Universal Robots PolyScope program: Pick_Place_demo.urp

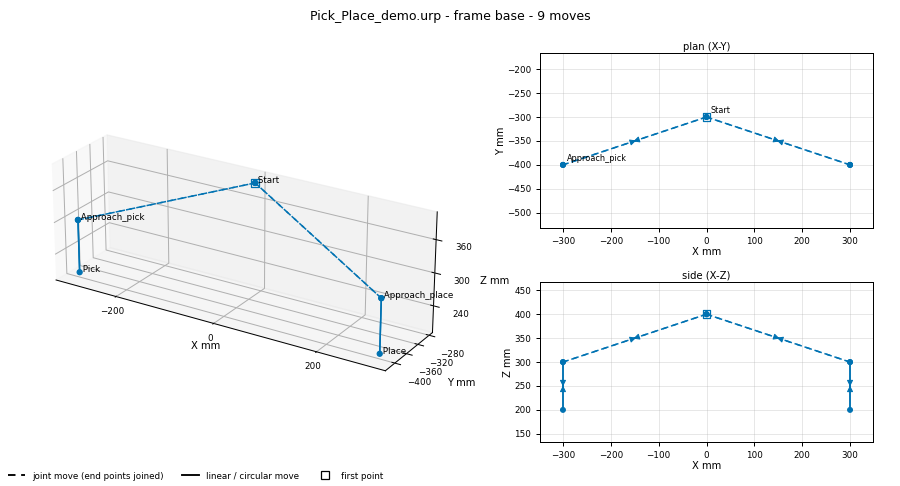
[picture p0: tool path of Pick_Place_demo.urp in frame base, 9 of 9 moves have a stored position in this frame; points joined in program order, loops and branches not executed]
Program Pick_Place_demo (installation=default directory=/programs/usbdisk createdIn=5.9.1.1031110 lastSavedIn=5.8.0.10253 robotSerialNumber=20205501179)
Calibrated DH parameters: a=[0.000177, -0.238276, -0.392216, 0.000101, -0.000031, 0]; d=[0.16274, -356.990158, 358.765662, -1.642182, 0.099681, 0.099622]; alpha=[1.570882, -0.000987, 0.009118, 1.568686, -1.570357, 0]; deltaTheta=[0, 0.976178, -0.934918, -0.041252, 0.000001, 0]
Robot Program (runOnlyOnce=false)
  MoveJ speed 60 deg/s, acceleration 80 deg/s^2 (useActiveTCP=true) feature=Base
    Waypoint Start: TCP in base x=0 y=-300 z=400 mm, rx=0 ry=3.1416 rz=0 rad; joints [-63.619, -58.456, -125.213, -86.33, 90, 26.381] deg
  Folder Pick
    MoveJ speed 60 deg/s, acceleration 80 deg/s^2 (useActiveTCP=true) feature=Base
      Waypoint Approach_pick: TCP in base x=-300 y=-400 z=300 mm, rx=0 ry=3.1416 rz=0 rad; joints [-111.408, -95.003, -113.354, -61.643, 90, -21.408] deg
    MoveL speed 250 mm/s, acceleration 1200 mm/s^2 (useActiveTCP=true) feature=Base
      Waypoint Pick: TCP in base x=-300 y=-400 z=200 mm, rx=0 ry=3.1416 rz=0 rad; joints [-111.408, -104.003, -120.574, -45.423, 90, -21.408] deg
      URCap 2FG Grip (OnRobot, OnRobot A/S) dataModel(twofg.external-grip.target-width=0.05, twofg.internal-grip.target-width=0.064, payload-weight=0.2)
      Waypoint Approach_pick: TCP in base x=-300 y=-400 z=300 mm, rx=0 ry=3.1416 rz=0 rad; joints [-111.408, -95.003, -113.354, -61.643, 90, -21.408] deg
    MoveJ speed 60 deg/s, acceleration 80 deg/s^2 (useActiveTCP=true) feature=Base
      Waypoint Start: TCP in base x=0 y=-300 z=400 mm, rx=0 ry=3.1416 rz=0 rad; joints [-63.619, -58.456, -125.213, -86.33, 90, 26.381] deg
  Folder Place
    MoveJ speed 60 deg/s, acceleration 80 deg/s^2 (useActiveTCP=true) feature=Base
      Waypoint Approach_place: TCP in base x=300 y=-400 z=300 mm, rx=0 ry=3.1416 rz=0 rad; joints [-37.668, -95.003, -113.354, -61.643, 90, 52.332] deg
    MoveL speed 250 mm/s, acceleration 1200 mm/s^2 (useActiveTCP=true) feature=Base
      Waypoint Place: TCP in base x=300 y=-400 z=200 mm, rx=0 ry=3.1416 rz=0 rad; joints [-37.668, -104.003, -120.574, -45.423, 90, 52.332] deg
      URCap 2FG Release (OnRobot, OnRobot A/S) dataModel(external_internal_action.index=0, twofg.external-grip.target-width=0.06, twofg.internal-grip.target-width=0.074)
      Waypoint Approach_place: TCP in base x=300 y=-400 z=300 mm, rx=0 ry=3.1416 rz=0 rad; joints [-37.668, -95.003, -113.354, -61.643, 90, 52.332] deg
    MoveJ speed 60 deg/s, acceleration 80 deg/s^2 (useActiveTCP=true) feature=Base
      Waypoint Start: TCP in base x=0 y=-300 z=400 mm, rx=0 ry=3.1416 rz=0 rad; joints [-63.619, -58.456, -125.213, -86.33, 90, 26.381] deg
  Folder Lamp
    Wait Sleep waitTime=2
    Popup Message (haltProgram=true message=End Program inputType=Text)
